ABB RobotStudio station: Locker.rspag

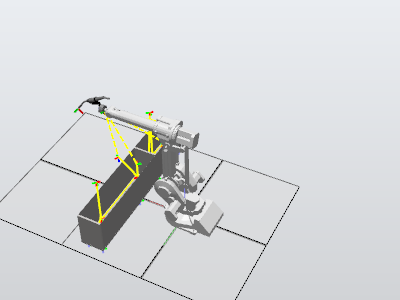
--- station ---
Station Project3 (saved by RobotStudio 23.2.10395.0)
Controller Controlador1
  mechanical unit ROB_1: IRB1410_5_144__01, 6 joints, base frame (0, 0, 0) mm
Layout (positions relative to the parent item):
  - IRB1410_5_144__01 [mechanism, from %ABB.RobotStudio.Models.IRB1410%\IRB1410_5_144_G_01.rslib] at (0, 0, 0) mm; joint values [0, 0, 0, 0, 0, 0] (rad or m)
  - AW_Gun_PSF_25 [mechanism, from %ABB.RobotStudio.Models.ArcWelding%\AW_Gun_PSF_25.rslib] at (955, 0, 1195) mm, rotated rx 0 ry 90 rz 0 deg
  - locker_3 [graphiccomponentgroup] at (100, -1200, -530) mm, rotated rx 0 ry -90 rz 0 deg
    - tapaext:1 [part] at (750.39, 2071.97, -584.08) mm, rotated rx 180 ry 0 rz 0 deg, size 431 x 20.5 x 281 mm
    - tapaext:2 [part] at (749.91, 271.97, -584.08) mm, size 431 x 20.5 x 281 mm
    - espaldar:1 [part] at (533.88, 1479.23, -530.21) mm, rotated rx 0 ry 0 rz -90 deg, size 1802 x 20.5 x 283 mm
    - lateral doblado:1 [part] at (740.39, 1171.97, -725.1) mm, rotated rx 90 ry 0 rz -90 deg, size 1798.9 x 20.5 x 429.4 mm
    - lateralsindoblar:1 [part] at (749.43, 1171.97, -444.7) mm, rotated rx 90 ry 0 rz -90 deg, size 1798.9 x 0.6 x 428.9 mm
    - tapnaint:1 [part] at (751.49, 870.87, -584.63) mm, size 431 x 20.5 x 279.9 mm
Attachment: AW_Gun_PSF_25 is attached to IRB1410_5_144__01 / Link6
Targets, tools, work objects and paths stored in the station and not in the controller backup, written as RAPID:
! task T_ROB1
MODULE Module1
  CONST jointtarget Home:=[[0,0,0,0,0,0],[9E+09,9E+09,9E+09,9E+09,9E+09,9E+09]];
  CONST robtarget Cajon1_Esq2:=[[804.076,-308.656,6.563],[0,0.5,0.866025404,0],[-1,-2,1,0],[9E+09,9E+09,9E+09,9E+09,9E+09,9E+09]];
  CONST robtarget Cajon1_limite1:=[[804.076,500,6.563],[0,0.5,0.866025404,0],[0,-1,1,0],[9E+09,9E+09,9E+09,9E+09,9E+09,9E+09]];
  CONST robtarget Cajon1_Esq1:=[[564.076,-308.656,6.563],[0,0.866025404,0.5,0],[-1,-1,1,0],[9E+09,9E+09,9E+09,9E+09,9E+09,9E+09]];
  CONST robtarget Cajon1_Giro1abajo:=[[804.076,500,6.563],[0,-0.573576436,0.819152045,0],[0,1,-2,0],[9E+09,9E+09,9E+09,9E+09,9E+09,9E+09]];
  CONST robtarget Cajon1_subida1:=[[804.076,500,600],[0,0.5,0.866025404,0],[0,-1,1,0],[9E+09,9E+09,9E+09,9E+09,9E+09,9E+09]];
  CONST robtarget Cajon1_Giro1arriba:=[[804.076,500,600],[0,-0.499999999,0.866025404,0],[0,0,-1,0],[9E+09,9E+09,9E+09,9E+09,9E+09,9E+09]];
  CONST robtarget Cajon1_Esq3:=[[750,850,6.563],[0,-0.573576436,0.819152044,0],[0,1,-2,0],[9E+09,9E+09,9E+09,9E+09,9E+09,9E+09]];
  CONST robtarget Cajon1_Esq4:=[[565,850,6.563],[0,0.866025404,-0.5,0],[0,0,-2,0],[9E+09,9E+09,9E+09,9E+09,9E+09,9E+09]];
  CONST robtarget Cajon1_Giro1abajo2:=[[804.076,800,6.563],[0,-0.499999999,0.866025404,0],[0,1,-2,0],[9E+09,9E+09,9E+09,9E+09,9E+09,9E+09]];
  CONST robtarget Cajon1_Fin:=[[565,50,6.563],[0,0.866025404,-0.5,0],[-1,0,-2,0],[9E+09,9E+09,9E+09,9E+09,9E+09,9E+09]];
  CONST robtarget Cajon1_Inicio:=[[564.076,50,6.563],[0,0.866025404,0.5,0],[0,-1,1,0],[9E+09,9E+09,9E+09,9E+09,9E+09,9E+09]];
  CONST robtarget Cajon1_Inicio_Ac2:=[[564.076,50,400],[0,0.866025404,0.5,0],[0,-1,1,0],[9E+09,9E+09,9E+09,9E+09,9E+09,9E+09]];
  CONST robtarget Cajon1_Inicio_Ac1:=[[800,50,600],[0,0.866025404,0.5,0],[0,-1,1,0],[9E+09,9E+09,9E+09,9E+09,9E+09,9E+09]];
  CONST robtarget Cajon1_Fin_Alej:=[[565,50,600],[0,0.866025404,-0.5,0],[-1,0,-2,0],[9E+09,9E+09,9E+09,9E+09,9E+09,9E+09]];
  CONST robtarget Cajon2_Inicio:=[[564.076,-700,6.563],[0,0.866025404,0.5,0],[-1,1,-1,0],[9E+09,9E+09,9E+09,9E+09,9E+09,9E+09]];
  CONST robtarget Cajon2_Esq1:=[[564.076,-905,6.563],[0,0.866025404,0.5,0],[-1,1,-1,0],[9E+09,9E+09,9E+09,9E+09,9E+09,9E+09]];
  CONST robtarget Cajon2_abajo1:=[[805,-670,6.563],[0,0.5,0.866025404,0],[-1,0,-1,0],[9E+09,9E+09,9E+09,9E+09,9E+09,9E+09]];
  CONST robtarget Cajon2_Esq2:=[[805,-905,6.563],[0,0.5,0.866025404,0],[-1,0,-1,0],[9E+09,9E+09,9E+09,9E+09,9E+09,9E+09]];
  CONST robtarget Cajon2_arriba1:=[[805,-670,700],[0,0.5,0.866025404,0],[-1,1,-2,0],[9E+09,9E+09,9E+09,9E+09,9E+09,9E+09]];
  CONST robtarget Cajon2_giro1:=[[805,-670,700],[0,-0.5,0.866025404,0],[-1,0,-2,0],[9E+09,9E+09,9E+09,9E+09,9E+09,9E+09]];
  CONST robtarget Cajon2_abajo2:=[[805,-580,6.563],[0,-0.5,0.866025404,0],[-1,0,-2,0],[9E+09,9E+09,9E+09,9E+09,9E+09,9E+09]];
  CONST robtarget Cajon2_Esq3:=[[805,-350,6.563],[0,-0.5,0.866025404,0],[-1,0,-2,0],[9E+09,9E+09,9E+09,9E+09,9E+09,9E+09]];
  CONST robtarget Cajon2_Esq4:=[[565,-350,6.563],[0,0.866025404,-0.5,0],[-1,0,-2,0],[9E+09,9E+09,9E+09,9E+09,9E+09,9E+09]];
  CONST robtarget Cajon2_Fin:=[[565,-580,6.563],[0,0.866025404,-0.5,0],[-1,0,-2,0],[9E+09,9E+09,9E+09,9E+09,9E+09,9E+09]];
  CONST robtarget Cajon2_Inicio_Ac:=[[564.076,-700,600],[0,0.866025404,0.5,0],[-1,1,-1,0],[9E+09,9E+09,9E+09,9E+09,9E+09,9E+09]];
  CONST robtarget Cajon2_Fin_Al:=[[565,-580,400],[0,0.866025404,-0.5,0],[-1,0,-2,0],[9E+09,9E+09,9E+09,9E+09,9E+09,9E+09]];
  CONST robtarget Cajon2_Fin_Al_2:=[[565,-580,400],[0,0.5,0.866025404,0],[-1,-1,-4,0],[9E+09,9E+09,9E+09,9E+09,9E+09,9E+09]];
  PROC Cajon_inferior()
    MoveAbsJ Home,v1000,z100,AW_Gun\WObj:=wobj0;
    MoveJ Cajon1_Inicio_Ac1,v1000,z100,AW_Gun\WObj:=wobj0;
    MoveL Cajon1_Inicio_Ac2,v1000,z100,AW_Gun\WObj:=wobj0;
    MoveL Cajon1_Inicio,v1000,z100,AW_Gun\WObj:=wobj0;
    MoveL Cajon1_Esq1,v1000,z100,AW_Gun\WObj:=wobj0;
    MoveL Cajon1_Esq2,v1000,z100,AW_Gun\WObj:=wobj0;
    MoveL Cajon1_limite1,v1000,z100,AW_Gun\WObj:=wobj0;
    MoveL Cajon1_subida1,v1000,z100,AW_Gun\WObj:=wobj0;
    MoveL Cajon1_Giro1arriba,v1000,z100,AW_Gun\WObj:=wobj0;
    MoveL Cajon1_Giro1abajo,v1000,z100,AW_Gun\WObj:=wobj0;
    MoveL Cajon1_Giro1abajo2,v1000,z100,AW_Gun\WObj:=wobj0;
    MoveL Cajon1_Esq3,v1000,z100,AW_Gun\WObj:=wobj0;
    MoveL Cajon1_Esq4,v1000,z100,AW_Gun\WObj:=wobj0;
    MoveL Cajon1_Fin,v1000,z100,AW_Gun\WObj:=wobj0;
    MoveL Cajon1_Fin_Alej,v1000,z100,AW_Gun\WObj:=wobj0;
    MoveAbsJ Home,v1000,z100,AW_Gun\WObj:=wobj0;
  ENDPROC
  PROC Cajon_superior()
    MoveAbsJ Home,v1000,z100,AW_Gun\WObj:=Workobject_1;
    MoveJ Cajon2_Inicio_Ac,v1000,z100,AW_Gun\WObj:=Workobject_1;
    MoveL Cajon2_Inicio,v1000,z100,AW_Gun\WObj:=Workobject_1;
    MoveL Cajon2_Esq1,v1000,z100,AW_Gun\WObj:=Workobject_1;
    MoveL Cajon2_Esq2,v1000,z100,AW_Gun\WObj:=Workobject_1;
    MoveL Cajon2_abajo1,v1000,z100,AW_Gun\WObj:=Workobject_1;
    MoveL Cajon2_arriba1,v1000,z100,AW_Gun\WObj:=Workobject_1;
    MoveJ Cajon2_giro1,v1000,z100,AW_Gun\WObj:=Workobject_1;
    MoveL Cajon2_abajo2,v1000,z100,AW_Gun\WObj:=Workobject_1;
    MoveL Cajon2_Esq3,v1000,z100,AW_Gun\WObj:=Workobject_1;
    MoveL Cajon2_Esq4,v1000,z100,AW_Gun\WObj:=Workobject_1;
    MoveL Cajon2_Fin,v1000,z100,AW_Gun\WObj:=Workobject_1;
    MoveL Cajon2_Fin_Al,v1000,z100,AW_Gun\WObj:=Workobject_1;
    MoveL Cajon2_Fin_Al_2,v1000,z100,AW_Gun\WObj:=Workobject_1;
    MoveAbsJ Home,v1000,z100,AW_Gun\WObj:=Workobject_1;
  ENDPROC
ENDMODULE

! task T_ROB1
MODULE CalibData
  PERS tooldata AW_Gun:=[TRUE,[[119.5,0,352],[0.890213743,0,0.455543074,0]],[1,[0,0,100],[1,0,0,0],0,0,0]];
  TASK PERS wobjdata Workobject_1:=[FALSE,TRUE,"",[[0,0,0],[1,0,0,0]],[[0,0,0],[1,0,0,0]]];
ENDMODULE


--- Controller Data/Controlador1/RAPID/TASK1/PROGMOD/Module1.mod ---
MODULE Module1
    !***********************************************************
    !
    ! M?dulo:  Module1
    !
    ! Descripción:
    !   <Introduzca la descripción aquí>
    !
    ! Autor: Andrago
    !
    ! Versión: 1.0
    !
    !***********************************************************


    !***********************************************************
    !
    ! Procedimiento Main
    !
    !   Este es el punto de entrada de su programa
    !
    !***********************************************************
    PROC main()
        !Add your code here
    ENDPROC
ENDMODULE
